{attribute 'GeneratedUsingTerminal: EL3356-0000-0017'}
{attribute addProperty BoxType "EL3356-0000-0017"}
{attribute addProperty Id "EtcSlaveTerminalBaseRMB_StatusAT %I*RMB_Status_C0E100AA7RMB_Value_INT32AT %I*RMB_Value_INT_E9189C4B4RMB_ControlAT %Q*RMB_Control_4997AEF64WcStateAT %I*WcState_9091E0EB2InfoDataAT %I*InfoData_32EB74EA10"}
{attribute addProperty CRC "776782056"}
{attribute addProperty Size "27"}
TYPE EL3356_2E4CC0E8 EXTENDS EtcSlaveTerminalBase :
STRUCT
	{attribute addProperty Name "RMB_Status"}
	RMB_Status : RMB_Status_C0E100AA;
	{attribute addProperty Name "RMB_Value_INT32"}
	RMB_Value_INT32 : RMB_Value_INT_E9189C4B;
	{attribute addProperty Name "RMB_Control"}
	RMB_Control : RMB_Control_4997AEF6;
	{attribute addProperty Name "WcState"}
	WcState : WcState_9091E0EB;
	{attribute addProperty Name "InfoData"}
	InfoData : InfoData_32EB74EA;
END_STRUCT
END_TYPE

(* stored: Version 1.2.0.0, ProductVersion 3.1.4024.9
   DUT EL3356_2E4CC0E8: Id {4a96b1e7-d6d7-4502-8739-eed011d3fc36} *)
